FUNCTION_BLOCK FB_Full
VAR_INPUT
    myInput         : LREAL;
END_VAR
VAR_OUTPUT
    myOutput        : BOOL := FALSE;
END_VAR
VAR
END_VAR

IF myInput > 0 THEN
    // FormatTrailingWhitespace
    IF myInput < 10 THEN                    
    	myOutput := TRUE;
	END_IF // FormatTabs
    // FormatInsertFinalNewline
END_IF

METHOD MyMethod : BOOL
VAR_INPUT
END_VAR
MyMethod := TRUE;
END_METHOD

PROPERTY Prop : BOOL
GET
Prop := TRUE;
END_GET
SET
END_SET
END_PROPERTY

END_FUNCTION_BLOCK

(* stored: Version 1.1.0.1, ProductVersion 3.1.4024.11
   POU FB_Full: Id {db56d684-bc10-4696-841c-dbe98e4576b1}, SpecialFunc None
   Method MyMethod: Id {300583ab-a978-412f-a94c-befedd5e1e5f}
   Property Prop: Id {8fd80566-d814-442c-877d-7ad2a8e592db}
   Get Get: Id {0e5e03b6-bf09-44cd-b757-f0cd34abbf52}
   Set Set: Id {8d674369-f153-4e28-9032-b7f6aa732966} *)
